PROGRAM MAIN
VAR
	XPlanarTable : FB_XPlanarModule;
	Initialize	 : BOOL; // Initialize the system
	Reset		 : BOOL; // Reset and Execute System
	Start		 : BOOL; // Run the system
	Halt		 : BOOL; // Avoid Disabling while spinning, otherwise physical sqauring of mover is required
	MachineState : (Startup,
		InitSystem,
		ResetSystem,
		Recover,
		Ready,
		Run,
		Disable);
	trig : R_TRIG;
END_VAR

//This project is a very simple "hello world" example for the APS4322 2-Tile starter kit.
//It is currently based on the XPlanarApplication library version 2.0.5 or greater.


//Keep all XPlanar motion system objects up to date every cycle
XPlanarTable.CyclicLogic();

// "Machine" Sequence
CASE MachineState OF
	Startup:	
		IF Initialize THEN
			Initialize := FALSE;
			MachineState := InitSystem;
		END_IF
	
	InitSystem:	
		IF XPlanarTable.Initialize() THEN
			MachineState := ResetSystem;
		END_IF
	
	ResetSystem:	
		IF Reset AND_THEN XPlanarTable.Reset() THEN
			Reset := FALSE;
			MachineState := Recover;
		END_IF
	
	Recover:	
		IF XPlanarTable.Recovery() THEN
			MachineState := Ready;
		END_IF
		
	Ready:
		IF Start THEN
			MachineState := Run;
		END_IF
	
	Run: 
		XPlanarTable.Execute();
	
	Disable:	
		IF XPlanarTable.Disable() THEN
			MachineState := 0;
		END_IF
END_CASE

IF Halt OR trig.Q THEN
	MachineState := Disable;
	Halt := FALSE;
END_IF

END_PROGRAM

(* stored: Version 1.1.0.1
   POU MAIN: Id {12228e0f-a5a3-4f5a-be0a-75fae71d01ff}, SpecialFunc None *)
